// TIA Portal V20 export
FUNCTION "V104" : Void   // FC21, FBD
{ S7_Optimized_Access := 'TRUE' }
// stored: SetENOAutomatically false
   VAR_TEMP
      Temp : "DigVal";
      Temp_1 : "DigVal";
      State : "Service_States";
   END_VAR
BEGIN

REGION Network 1: Channel input
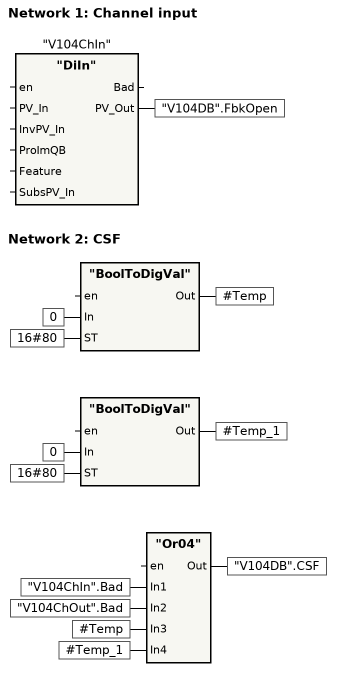
   "V104ChIn"(PV_Out => "V104DB".FbkOpen);   // "DiIn"
END_REGION

REGION Network 2: CSF
   "BoolToDigVal"(In := 0, ST := 16#80, Out => #Temp);
   "BoolToDigVal"(In := 0, ST := 16#80, Out => #Temp_1);
   "Or04"(In1 := "V104ChIn".Bad, In2 := "V104ChOut".Bad, In3 := #Temp, In4 := #Temp_1, Out => "V104DB".CSF);
END_REGION

REGION Network 3: VlvAn Intlock
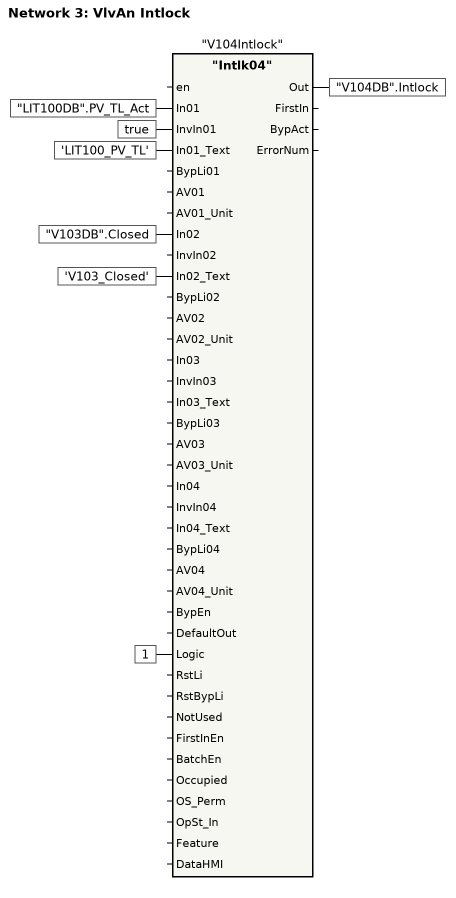
   "V104Intlock"(In01 := "LIT100DB".PV_TL_Act,   // "Intlk04"
                 InvIn01 := true,
                 In01_Text := 'LIT100_PV_TL',
                 In02 := "V103DB".Closed,
                 In02_Text := 'V103_Closed',
                 Logic := 1,
                 Out => "V104DB".Intlock);
END_REGION

REGION Network 4: VlvAnL
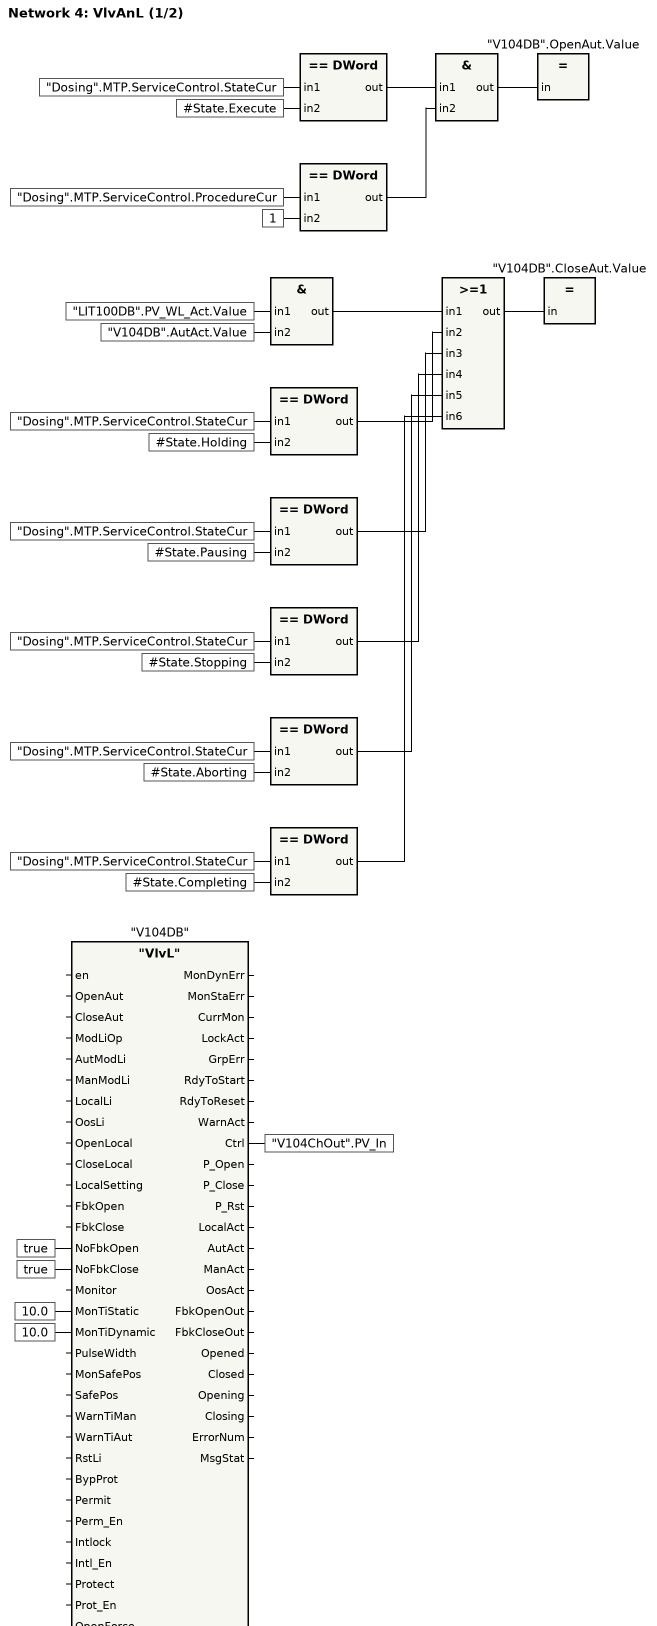
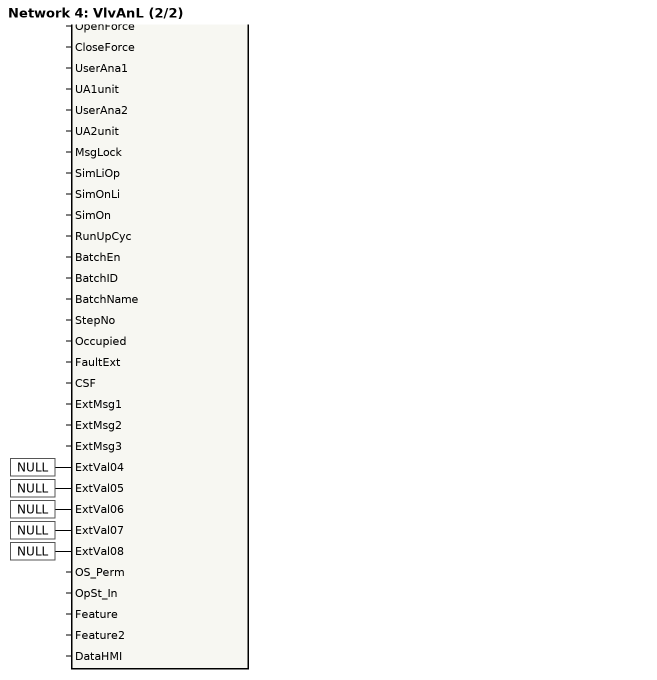
   "V104DB".OpenAut.Value := ("Dosing".MTP.ServiceControl.StateCur = #State.Execute) AND ("Dosing".MTP.ServiceControl.ProcedureCur = 1);
   "V104DB".CloseAut.Value := ("LIT100DB".PV_WL_Act.Value AND "V104DB".AutAct.Value) OR ("Dosing".MTP.ServiceControl.StateCur = #State.Holding) OR ("Dosing".MTP.ServiceControl.StateCur = #State.Pausing) OR ("Dosing".MTP.ServiceControl.StateCur = #State.Stopping) OR ("Dosing".MTP.ServiceControl.StateCur = #State.Aborting) OR ("Dosing".MTP.ServiceControl.StateCur = #State.Completing);
   "V104DB"(NoFbkOpen := true,   // "VlvL"
            NoFbkClose := true,
            MonTiStatic := 10.0,
            MonTiDynamic := 10.0,
            ExtVal04 := NULL,
            ExtVal05 := NULL,
            ExtVal06 := NULL,
            ExtVal07 := NULL,
            ExtVal08 := NULL,
            Ctrl => "V104ChOut".PV_In);
END_REGION

REGION Network 5: MTP
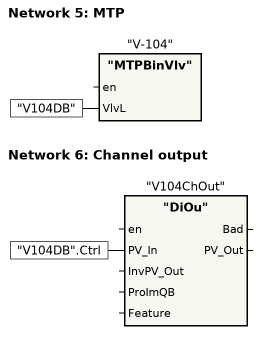
   "V-104"(VlvL := "V104DB");   // "MTPBinVlv"
END_REGION

REGION Network 6: Channel output
   "V104ChOut"(PV_In := "V104DB".Ctrl);   // "DiOu"
END_REGION
END_FUNCTION
